TYPE U_MOVER_INFO :
UNION
  stInfo              : ARRAY[1..MAX_MOVER] OF ST_MOVER_INFO;

  byInfo    AT %Q*    : ARRAY[1..MAX_MOVER] OF
                        ARRAY[1..SIZEOF(ST_MOVER_INFO)] OF BYTE;
END_UNION
END_TYPE

(* stored: Version 1.1.0.1, ProductVersion 3.1.4026.12
   DUT U_MOVER_INFO: Id {fa883135-7ff2-4ea6-a920-efdb21a2e09c} *)
